// TwinCAT 3 PLC project PLC1
// Title: Actuator
// Company: Promise Robotics
// ProjectVersion: 0.0.5
// ProgramVersion: 3.1.4026.16
// libraries:
//   DigitalInput, * (Promise Robotics)
//   DigitalOutput, * (Promise Robotics)
//   Tc2_Standard, * (Beckhoff Automation GmbH)
//   Tc2_System, * (Beckhoff Automation GmbH)
// project tree:
//   POUs/ E_ActuatorState.TcDUT, FB_Actuator.TcPOU, FB_MultiActuator_NoFeedback.TcPOU, FB_Actuator_NoFeedback.TcPOU, ITF_Actuator.TcIO

// ---- POUs/E_ActuatorState.TcDUT
{attribute 'qualified_only'}
{attribute 'strict'}
{attribute 'to_string'}
TYPE E_ActuatorState :
(
	Retract,
	Advance
);
END_TYPE

// ---- POUs/ITF_Actuator.TcIO
INTERFACE ITF_Actuator

METHOD Advance
VAR_INPUT
END_VAR
END_METHOD

PROPERTY P_Advanced : BOOL
GET
END_GET
END_PROPERTY

PROPERTY P_OperatorControl : BOOL
GET
END_GET
SET
END_SET
END_PROPERTY

PROPERTY P_OperatorValue : E_ActuatorState
GET
END_GET
SET
END_SET
END_PROPERTY

PROPERTY P_Retracted : BOOL
GET
END_GET
END_PROPERTY

METHOD Retract
VAR_INPUT
END_VAR
END_METHOD

END_INTERFACE

// ---- POUs/FB_Actuator.TcPOU
FUNCTION_BLOCK FB_Actuator IMPLEMENTS ITF_Actuator
VAR
	AdvanceBit		: BOOL := FALSE;
	RetractBit		: BOOL := FALSE;
	
	AdvanceTimer	: TON;
	RetractTimer	: TON;
	
	{ attribute 'TcHmiSymbol.AddSymbol' }
	OperatorControl	: BOOL := FALSE; //HMI Operator Control (Actuator state reverts to original state when out of Op control)
	OpControlFTRIG	: F_TRIG;
	
	{ attribute 'TcHmiSymbol.AddSymbol' }
	OperatorValue	: E_ActuatorState; //HMI Operator Value
	HeldValue		: E_ActuatorState;
	
	HardwareOverride	: BOOL; //For engineering actuator overriding
	OverrideValue		: E_ActuatorState; //Override Value
END_VAR

VAR_INPUT
	AdvancedIN		: FB_DigitalInput;
	RetractedIN		: FB_DigitalInput;
	AdvanceOUT		: FB_DigitalOutput;
	RetractOUT		: FB_DigitalOutput;
END_VAR

AdvanceOUT();
RetractOUT();

AdvancedIN();
RetractedIN();

AdvanceTimer(IN := AdvanceBit, PT := T#0.06S);
AdvanceOUT.SetOutput(AdvanceTimer.Q);

RetractTimer(IN := RetractBit, PT := T#0.06S);
RetractOUT.SetOutput(RetractTimer.Q);

//Retain value prior to going into operator control
OpControlFTRIG(CLK := OperatorControl);
IF OpControlFTRIG.Q THEN
	IF HeldValue = E_ActuatorState.Advance THEN
		Advance();
	ELSIF HeldValue = E_ActuatorState.Retract THEN
		Retract();
	END_IF
END_IF

IF NOT OperatorControl AND NOT HardwareOverride AND AdvancedIN.P_Value THEN
	OperatorValue 	:= E_ActuatorState.Advance;
	OverrideValue	:= E_ActuatorState.Advance;
	HeldValue 		:= E_ActuatorState.Advance;
ELSIF NOT OperatorControl AND NOT HardwareOverride AND RetractedIN.P_Value THEN
	OperatorValue 	:= E_ActuatorState.Retract;
	OverrideValue	:= E_ActuatorState.Retract;
	HeldValue 		:= E_ActuatorState.Retract;
END_IF

IF OperatorControl THEN
	IF OperatorValue = E_ActuatorState.Advance THEN
		Advance();
	ELSIF OperatorValue = E_ActuatorState.Retract THEN
		Retract();
	END_IF
END_IF

IF HardwareOverride THEN
	IF OverrideValue = E_ActuatorState.Advance THEN
		Advance();
	ELSIF OverrideValue = E_ActuatorState.Retract THEN
		Retract();
	END_IF
END_IF

METHOD Advance
RetractOUT.SetOutput(FALSE);
RetractBit := FALSE;
AdvanceBit := TRUE;
END_METHOD

PROPERTY P_Advanced : BOOL
GET
P_Advanced := AdvancedIN.P_Value;
END_GET
END_PROPERTY

PROPERTY P_OperatorControl : BOOL
GET
P_OperatorControl := OperatorControl;
END_GET
SET
OperatorControl := P_OperatorControl;
END_SET
END_PROPERTY

PROPERTY P_OperatorValue : E_ActuatorState
GET
P_OperatorValue := OperatorValue;
END_GET
SET
OperatorValue := P_OperatorValue;
END_SET
END_PROPERTY

PROPERTY P_Retracted : BOOL
GET
P_Retracted := RetractedIN.P_Value;
END_GET
END_PROPERTY

METHOD Retract
AdvanceOUT.SetOutput(FALSE);
RetractBit := TRUE;
AdvanceBit := FALSE;
END_METHOD

END_FUNCTION_BLOCK

// ---- POUs/FB_MultiActuator_NoFeedback.TcPOU
FUNCTION_BLOCK FB_MultiActuator_NoFeedback
VAR_GENERIC CONSTANT
	LenActuators : UDINT := 1;
END_VAR
VAR
	Actuator : ARRAY[0..LenActuators-1] OF FB_Actuator_NoFeedback;
END_VAR

END_FUNCTION_BLOCK

// ---- POUs/FB_Actuator_NoFeedback.TcPOU
FUNCTION_BLOCK FB_Actuator_NoFeedback
VAR
	AdvanceOUT		: FB_DigitalOutput;
	RetractOUT		: FB_DigitalOutput;
	
	AdvanceBit			: BOOL := FALSE;
	RetractBit			: BOOL := FALSE;
	
	Advanced		: BOOL := FALSE;
	Retracted		: BOOL := FALSE;
	
	AdvanceTimer	: TON;
	RetractTimer	: TON;
END_VAR

AdvanceOUT();
RetractOUT();

AdvanceTimer(IN := AdvanceBit, PT := T#0.06S);
AdvanceOUT.SetOutput(AdvanceTimer.Q);
Advanced := AdvanceOUT.P_Output;

RetractTimer(IN := RetractBit, PT := T#0.06S);
RetractOUT.SetOutput(RetractTimer.Q);
Retracted := RetractOUT.P_Output;

METHOD PUBLIC Advance : BOOL
RetractOUT.SetOutput(FALSE);
RetractBit := FALSE;
Advance := TRUE;
END_METHOD

PROPERTY P_Advanced : BOOL
GET
P_Advanced := Advanced;
END_GET
END_PROPERTY

PROPERTY P_Retracted : BOOL
GET
P_Retracted := Retracted;
END_GET
END_PROPERTY

METHOD PUBLIC Retract : BOOL
AdvanceOUT.SetOutput(FALSE);
Retract := TRUE;
AdvanceBit := FALSE;
END_METHOD

END_FUNCTION_BLOCK
